FUNCTION F_ServoDirection : MC_DIRECTION
VAR_INPUT
	ServoMoveType		: E_ServoMoveType;
END_VAR

CASE ServoMoveType OF
	eServoMoveType_MODULO_SHORTEST_PATH : 
		F_ServoDirection := MC_Shortest_Way;
	eServoMoveType_MODULO_POSITIVE : 
		F_ServoDirection := MC_Positive_Direction;
	eServoMoveType_MODULO_NEGATIVE : 
		F_ServoDirection := MC_Negative_Direction;
END_CASE

END_FUNCTION

(* stored: Version 1.1.0.1, ProductVersion 3.1.4024.3
   POU F_ServoDirection: Id {af1de19d-7c46-4d50-83cf-2ad09cf4a250}, SpecialFunc None *)
